(* IEC 61131-3 sources: InfiniteStateMachine/st/library_information, 2 files *)

(* ---- getlibversion-GetLibVersion.st ---- *)
(* --- Interface --- *)
// This function has been automatically generated from the project information.
FUNCTION GetLibVersion : VERSION
VAR_INPUT

END_VAR
(* --- Implementation --- *)
GetLibVersion.uiMajor := 0;
GetLibVersion.uiMinor := 1;
GetLibVersion.uiServicePack := 1;
GetLibVersion.uiPatch := 1;

(* ---- islibreleased-IsLibReleased.st ---- *)
(* --- Interface --- *)
// This function has been automatically generated from the project information.
FUNCTION IsLibReleased : BOOL
VAR_INPUT

END_VAR
(* --- Implementation --- *)
IsLibReleased := FALSE;
